Omron CX-Programmer project NewProject (CX-Programmer 9.61)

# PLC NewPLC1: CJ1M CPU11

## Global symbols (name address type ; comment)
0.00 BOOL  ; Start
100.00 BOOL  ; M1
100.01 BOOL  ; M2
10.00 BOOL  ; G_P
10.01 BOOL  ; R
10.02 BOOL  ; G
10.03 BOOL  ; R_P
10.04 BOOL  ; Y
T0000 BOOL  ; Tim1
T0001 BOOL  ; Tim2
T0002 BOOL  ; Tim3
T0003 BOOL  ; Tim4
T0004 BOOL  ; Tim5
T0005 BOOL  ; Tim6
T0006 BOOL  ; Tim7

## Program NewProgram1 (cyclic task 0)

### Section Section1

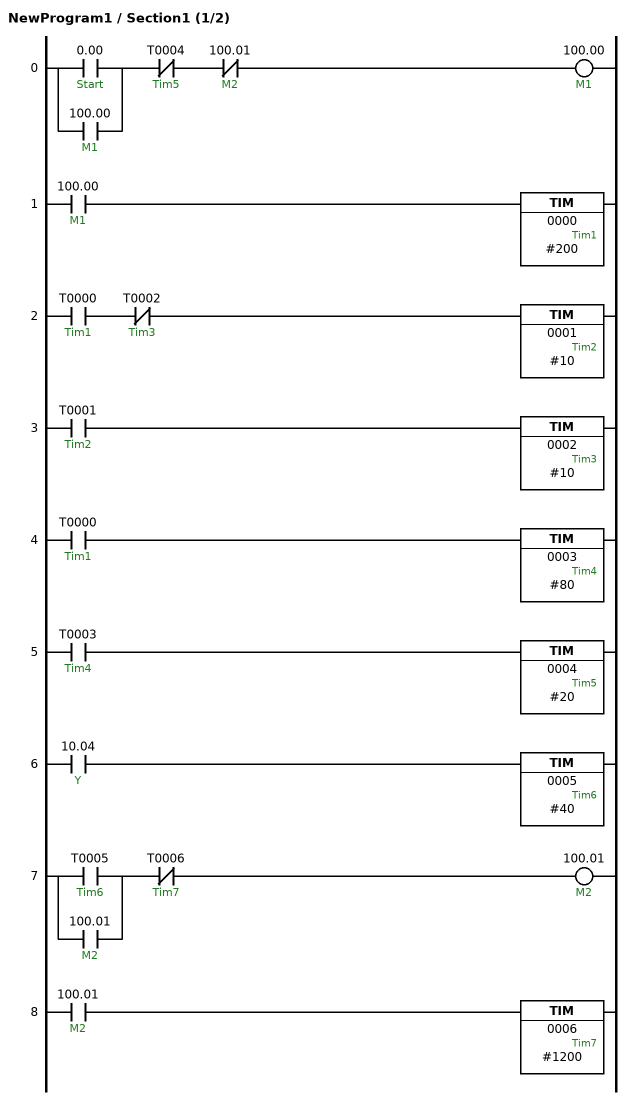
; rung 0
LD 0.00  ; Start
OR 100.00  ; M1
ANDNOT T0004  ; Tim5
ANDNOT 100.01  ; M2
OUT 100.00  ; M1
; rung 1
LD 100.00  ; M1
TIM 0000 #200  ; Tim1
; rung 2
LD T0000  ; Tim1
ANDNOT T0002  ; Tim3
TIM 0001 #10  ; Tim2
; rung 3
LD T0001  ; Tim2
TIM 0002 #10  ; Tim3
; rung 4
LD T0000  ; Tim1
TIM 0003 #80  ; Tim4
; rung 5
LD T0003  ; Tim4
TIM 0004 #20  ; Tim5
; rung 6
LD 10.04  ; Y
TIM 0005 #40  ; Tim6
; rung 7
LD T0005  ; Tim6
OR 100.01  ; M2
ANDNOT T0006  ; Tim7
OUT 100.01  ; M2
; rung 8
LD 100.01  ; M2
TIM 0006 #1200  ; Tim7

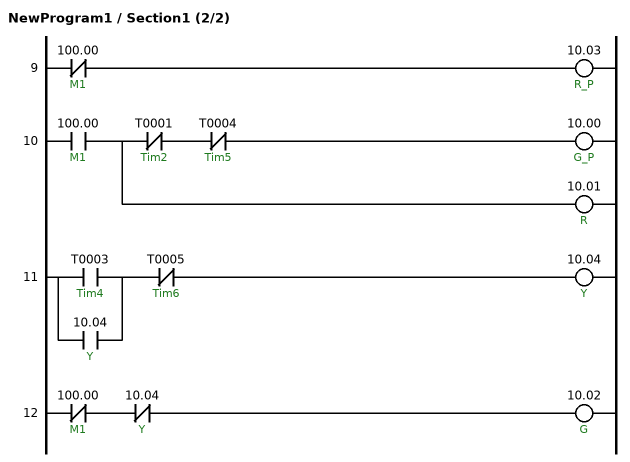
; rung 9
LDNOT 100.00  ; M1
OUT 10.03  ; R_P
; rung 10
LD 100.00  ; M1
OUT TR0
ANDNOT T0001  ; Tim2
ANDNOT T0004  ; Tim5
OUT 10.00  ; G_P
LD TR0
OUT 10.01  ; R
; rung 11
LD T0003  ; Tim4
OR 10.04  ; Y
ANDNOT T0005  ; Tim6
OUT 10.04  ; Y
; rung 12
LDNOT 100.00  ; M1
ANDNOT 10.04  ; Y
OUT 10.02  ; G

### Section END
; rung 0
END(001)